// TwinCAT 3 PLC project PLC_BatchControl
// ProgramVersion: 3.1.4026.24
// libraries:
//   Tc2_Standard, * (Beckhoff Automation GmbH)
//   Tc2_System, * (Beckhoff Automation GmbH)
// project tree:
//   / PlcTask.TcTTO
//   POUs/ MAIN.TcPOU
// real-time tasks:
//   TASK PlcTask: cycle T#10ms, priority 20, ADS port 350

CONFIGURATION PLC_BatchControl
    RESOURCE PLC ON TwinCAT3
        TASK PlcTask(INTERVAL := T#10ms, PRIORITY := 20);
        PROGRAM MAIN WITH PlcTask : MAIN;
    END_RESOURCE
END_CONFIGURATION

// ---- POUs/MAIN.TcPOU
PROGRAM MAIN
VAR
	systemActive: BOOL;
	startMix: BOOL;
	mixTimer: TON;
	startFill: BOOL;
	counterA: CTU;
	counterB: CTU;
	tankLevelA: BOOL;
	tankLevelB: BOOL;
	valveA: BOOL;
	valveB: BOOL;
	mixerMotor: BOOL;
	
END_VAR

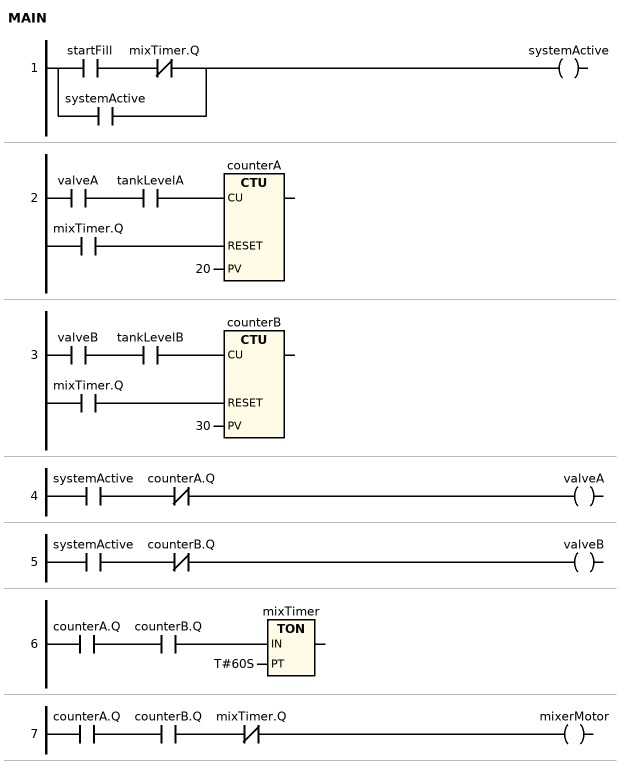
// NETWORK 1
systemActive := startFill AND NOT mixTimer.Q OR systemActive;

// NETWORK 2
counterA(CU := valveA AND tankLevelA, RESET := mixTimer.Q, PV := 20); // CTU

// NETWORK 3
counterB(CU := valveB AND tankLevelB, RESET := mixTimer.Q, PV := 30); // CTU

// NETWORK 4
valveA := systemActive AND NOT counterA.Q;

// NETWORK 5
valveB := systemActive AND NOT counterB.Q;

// NETWORK 6
mixTimer(IN := counterA.Q AND counterB.Q, PT := T#60S); // TON

// NETWORK 7
mixerMotor := (counterA.Q AND counterB.Q) AND NOT mixTimer.Q;

END_PROGRAM
